// SIMATIC S7-200 project (STEP 7-Micro/WIN), CPU 224 CN REL 02.01

ORGANIZATION_BLOCK 主程序:OB1
TITLE=当操作员按下触发数据更新按钮时，系统会将运动参数存储区中的数据（如目标速度或位置）更新到运动参数目标地址指向的位置，为后续运动提供参数基础。
// 当生产需要传送带移动到特定位置时，运动启用标志会被置位，且运动启动脉冲产生上升沿触发信号，系统执行相应的运动控制。
// 当需要更新传送带当前位置时，若装载启用信号被置位，且装载触发脉冲产生上升沿，系统会将新的位置数据装载到当前位置。
// 运行状态通过指示灯实时显示。当运行控制信号为真时，运行指示灯点亮，提示传送带正在工作。
// 若出现异常情况，当报警触发信号为真时，报警指示灯点亮，提醒操作员检查问题
BEGIN
Network 1
LD     M1.1
MOVD   VD300, VD43
-D     +48, VD43
Network 2 // 网络标题
// 网络注释
LD     SM0.0
=      L60.0
LD     M0.0
=      L63.7
LD     M0.1
=      L63.6
LD     L60.0
CALL   PTO0_CTRL:SBR1, L63.7, L63.6, V80.0, VB100, VD150
Network 3
LD     M0.2
=      L60.0
LD     M0.3
EU
=      L63.7
LD     L60.0
CALL   PTO0_RUN:SBR2, L63.7, VB102, M0.4, V80.1, VB101, VB103, VB104, VD154
Network 4
LD     M0.5
=      L60.0
LD     M0.6
EU
=      L63.7
LD     L60.0
CALL   PTO0_LDPOS:SBR4, L63.7, VD158, V80.2, VB105, VD162
Network 5
LD     M0.7
=      Q2.0
Network 6
LD     M1.0
=      Q2.5
END_ORGANIZATION_BLOCK

// SBR1: protected block, not included

// SBR2: protected block, not included

// SBR3: protected block, not included

// SBR4: protected block, not included

// (further data pages could not be read)
